PROGRAM MonitoringTheSoilTask
VAR
	Timer: TON;
	state: INT;
	Moisture: REAL;
	Temp: REAL;
	WaterRequired: BOOL;
END_VAR

0

CASE state OF
	0:// Initial position
	Moisture :=50;
	Temp := 25;
	state :=1;
	
	1: //ReadSensors
	Moisture:= Moisture - 1
	IF Moisture < 0 THEN Moisture :=0 END_IF;
	Temp := Temp;
	state := 2;
	 
	2://UpdateGVL
	WaterRequired := (Moisture <30 AND Temp > 20 );
	State:=1;

	
	
	
	
END_CASE

END_PROGRAM

(* stored: Version 1.1.0.1, ProductVersion 3.1.4024.15
   POU MonitoringTheSoilTask: Id {e84dcc4b-2fdc-469e-92e0-8f395adb38ff}, SpecialFunc None *)
